{region '#Template'}
	{attribute 'Category' := 'Universal'}
	{attribute 'Version' := '0.0.1.0'}
	{attribute 'Tags' := 'Universal, Control, PID, Loop'}
	{attribute 'Description' := 'Regler	// Controller'}
{endregion}
FUNCTION_BLOCK FB_BA_PID EXTENDS FB_BA_View
VAR_INPUT
	bEn						: BOOL;
	fW						: REAL;
	fX						: REAL;
	bSync					: BOOL;
	fSync					: REAL;
END_VAR
VAR_OUTPUT
	fY						: REAL;
	fMax					: REAL;
	fMin					: REAL;	
END_VAR
VAR_INPUT CONSTANT		 
	Ctrl					: FB_BA_Loop;	
END_VAR

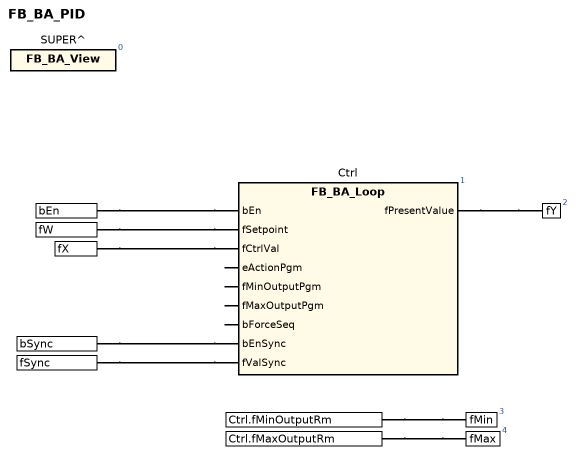
SUPER^(); // FB_BA_View
Ctrl(bEn := bEn, fSetpoint := fW, fCtrlVal := fX, bEnSync := bSync, fValSync := fSync); // FB_BA_Loop
fY := Ctrl.fPresentValue;
fMin := Ctrl.fMinOutputRm;
fMax := Ctrl.fMaxOutputRm;

METHOD FB_init : BOOL
VAR_INPUT
	bInitRetains : BOOL; // if TRUE, the retain variables are initialized (warm start / cold start)
	bInCopyCode : BOOL;  // if TRUE, the instance afterwards gets moved into the copy code (online change)
END_VAR
Ctrl.iParent				:= THIS^;
Ctrl.iLabel					:= LblUniControl.PID_Ctrl; 
Ctrl.sObjectName			:= '{Idx=01}';
Ctrl.eOpMode				:= BA2_Param.nLoop_DefOpMode;								 	 										 
Ctrl.eOutputUnit			:= E_BA_Unit.eOther_Percent;
Ctrl.eActionRm				:= E_BA_Action.eReverse;
Ctrl.fProportionalConstant	:= 3;
Ctrl.fIntegralConstant		:= 180;
Ctrl.fDerivativeConstant	:= 0;
Ctrl.fMaxOutputRm 			:= 100;
Ctrl.fMinOutputRm			:= 0;
Ctrl.fCOVIncrement			:= 0;
Ctrl.nDampConstant			:= 0;
Ctrl.fNeutralZone			:= 0;
Ctrl.stStepDelay.nDown		:= 0;
Ctrl.stStepDelay.nUp		:= 0;
END_METHOD

END_FUNCTION_BLOCK

(* stored: Version 1.1.0.1, ProductVersion 3.1.4024.6
   POU FB_BA_PID: Id {3bf0c719-1523-4ed5-84c9-9ea0145135eb}, SpecialFunc None
   Method FB_init: Id {f55e5579-1204-45ad-8aea-48ef49401ac5} *)
